{attribute 'qualified_only'}
VAR_GLOBAL		
	AI_1 AT %I*: INT;// Analogeingang AI 1
	AI_2 AT %I*: INT;// Analogeingang AI 2
	
	AQ_1 AT %Q*: INT;// Analogausgang AQ 1
	AQ_2 AT %Q*: INT;// Analogausgang AQ 2
END_VAR

(* stored: Version 1.1.0.1, ProductVersion 3.1.4022.7
   GVL Plc_AN: Id {cd2b667e-56d6-422c-ab59-5b92b8a35891} *)
